{attribute 'pack_mode' := '1'}
TYPE ST_EnableStationDataIn :
STRUCT
	sCellID						: STRING(30);
	sID							: STRING(30);
	bPresent					: BOOL;
END_STRUCT
END_TYPE

(* stored: Version 1.1.0.1, ProductVersion 3.1.4024.5
   DUT ST_EnableStationDataIn: Id {26e52b7c-91c7-406d-99e3-a04bab75290f} *)
